Staubli VAL3: SaveAction.pgx

public program SaveAction(bool& x_bRes (dimensions=1))
  local num l_nNum
  local num l_nX
  local string l_sFileName
  local string l_sSBuff
begin


  //参数初始化
  x_bRes=false
  l_sFileName="Disk://Txt/Action.txt"


  //关闭所有文件
  call FileDir:CloseAllFile()


  //文件是否可以打开
  nFileID=$fileOpen(l_sFileName,"w")
  if nFileID<0 or nFileID>9
    return
  endIf


  for l_nNum=1 to 50
    l_sSBuff=toString("",l_nNum)+"="
    for l_nX=0 to 11
      l_sSBuff=l_sSBuff+toString("",nAction[l_nNum,l_nX,0])+","+toString(".2",nAction[l_nNum,l_nX,1])+";"
    endFor
    if $fileSet(nFileID,l_sSBuff,1)!=1
      return
    endIf
  endFor

  call FileDir:CloseAllFile()

  x_bRes=true

end
